# EPICS autosave request: soft_iocs/galil_DMC/iocBoot/iocgalil_DMC_E05/GalilTest_18ID_DMC_E05Positions.req
$(P)33.DVAL
$(P)34.DVAL
$(P)35.DVAL
$(P)36.DVAL
$(P)37.DVAL
$(P)38.DVAL
$(P)39.DVAL
$(P)40.DVAL
